// TwinCAT 3 PLC project CustomGenericDataType
// Title: TwinCAT Custom Generic Data Types
// Company: FisoThemes
// Author: Goodwill Mzumala
// ProjectVersion: 1.0.0.0
// Description: Library created to handle data in TwinCAT generically. Useful for overloading or creating multitype arrays.
// ProgramVersion: 3.1.4023.0
// libraries:
//   Tc2_Standard, * (Beckhoff Automation GmbH)
//   Tc2_System, * (Beckhoff Automation GmbH)
//   Tc3_Module, * (Beckhoff Automation GmbH)
// project tree:
//   DUTs/ ST_Arg_Pointer.TcDUT, ST_Arg.TcDUT
//   / PlcTask.TcTTO
//   POUs/Arguments/Bit/ F_BYTE_ARG.TcPOU, F_DWORD_ARG.TcPOU, F_LWORD_ARG.TcPOU, F_WORD_ARG.TcPOU
//   POUs/Arguments/Date/ F_DATE_ARG.TcPOU, F_DT_ARG.TcPOU, F_TOD_ARG.TcPOU
//   POUs/Arguments/Int/ F_DINT_ARG.TcPOU, F_INT_ARG.TcPOU, F_LINT_ARG.TcPOU, F_SINT_ARG.TcPOU, F_UDINT_ARG.TcPOU, F_UINT_ARG.TcPOU, F_ULINT_ARG.TcPOU, F_USINT_ARG.TcPOU
//   POUs/Arguments/Other/ F_ANY_ARG.TcPOU, F_PVOID_ARG.TcPOU
//   POUs/Arguments/Real/ F_LREAL_ARG.TcPOU, F_REAL_ARG.TcPOU
//   POUs/Arguments/String/ F_STRING_ARG.TcPOU, F_WSTRING_ARG.TcPOU
//   POUs/Arguments/Time/ F_LTIME_ARG.TcPOU, F_TIME_ARG.TcPOU
//   POUs/Examples/Example 1 - Generic Use Case/ P_Example_1.TcPOU
//   POUs/Examples/Example 2 - Dynamic Array Use Case/Files/ FB_Dynamic_Array.TcPOU, T_DynamicArrayDataType.TcDUT
//   POUs/Examples/Example 2 - Dynamic Array Use Case/ P_Example_2.TcPOU
//   POUs/ MAIN.TcPOU
//   POUs/Return Values/Bit/ F_BYTE_RTN.TcPOU, F_DWORD_RTN.TcPOU, F_LWORD_RTN.TcPOU, F_WORD_RTN.TcPOU
//   POUs/Return Values/Date/ F_DATE_RTN.TcPOU, F_DT_RTN.TcPOU, F_TOD_RTN.TcPOU
//   POUs/Return Values/Int/ F_DINT_RTN.TcPOU, F_INT_RTN.TcPOU, F_LINT_RTN.TcPOU, F_SINT_RTN.TcPOU, F_UDINT_RTN.TcPOU, F_UINT_RTN.TcPOU, F_ULINT_RTN.TcPOU, F_USINT_RTN.TcPOU
//   POUs/Return Values/Other/ F_PVOID_RTN.TcPOU
//   POUs/Return Values/Real/ F_LREAL_RTN.TcPOU, F_REAL_RTN.TcPOU
//   POUs/Return Values/String/ F_STRING_RTN.TcPOU, F_WSTRING_RTN.TcPOU
//   POUs/Return Values/Time/ F_LTIME_RTN.TcPOU, F_TIME_RTN.TcPOU
// real-time tasks:
//   TASK PlcTask: cycle T#10ms, priority 20, ADS port 350

CONFIGURATION CustomGenericDataType
    RESOURCE PLC ON TwinCAT3
        TASK PlcTask(INTERVAL := T#10ms, PRIORITY := 20);
        PROGRAM MAIN WITH PlcTask : MAIN;
    END_RESOURCE
END_CONFIGURATION

// ---- DUTs/ST_Arg_Pointer.TcDUT
(* Collection of pointers for F_ANY_ARG. *)
TYPE INTERNAL ST_Arg_Pointer :
STRUCT
    pBool			: POINTER TO BOOL;
    pByte			: POINTER TO BYTE;
    pWord			: POINTER TO WORD;
    pDWord			: POINTER TO DWORD;
    pLWord			: POINTER TO LWORD;
    pSint			: POINTER TO SINT;
    pInt			: POINTER TO INT;
    pDint			: POINTER TO DINT;
    pLint			: POINTER TO LINT;
    pUSint			: POINTER TO USINT;
    pUInt			: POINTER TO UINT;
    pUDint			: POINTER TO UDINT;
    pULint			: POINTER TO ULINT;
    pReal			: POINTER TO REAL;
    pLReal			: POINTER TO LREAL;
    pString			: POINTER TO STRING;
    pWString		: POINTER TO WSTRING;
    pTime			: POINTER TO TIME;
    pDate			: POINTER TO DATE;
    pDate_And_Time	: POINTER TO DATE_AND_TIME;
    pTime_Of_Day	: POINTER TO TIME_OF_DAY;
    pPointer		: PVOID;
	pLTime 			: POINTER TO LTIME;
END_STRUCT
END_TYPE

// ---- DUTs/ST_Arg.TcDUT
(* Generic data type used for Programs/Functions/Function Blocks. *)
TYPE ST_Arg EXTENDS __SYSTEM.AnyType :
STRUCT
	sValue : T_MaxString; 	// Data of parameter as a string for easy convertion.
END_STRUCT
END_TYPE

// ---- POUs/Examples/Example 2 - Dynamic Array Use Case/Files/T_DynamicArrayDataType.TcDUT
TYPE T_DynamicArrayDataType : ST_Arg; END_TYPE

// ---- POUs/MAIN.TcPOU
PROGRAM MAIN
VAR
	
END_VAR

P_Example_1();
P_Example_2();

END_PROGRAM

// ---- POUs/Examples/Example 1 - Generic Use Case/P_Example_1.TcPOU
PROGRAM P_Example_1
VAR
	stArg 	: ARRAY[0..5] OF ST_Arg;
	
	Numeric_Type 		: INT := 20;
	User_Defined_Type	: TON := (PT := T#10S);
	
	rtnInteger 	: INT;
	rtnPointer 	: POINTER TO TON;
	
END_VAR

// Store 
stArg[0] := F_ANY_ARG(Numeric_Type);
stArg[1] := F_INT_ARG(1);
stArg[2] := F_REAL_ARG(12.442);
stArg[3] := F_STRING_ARG('Cats');
stArg[4] := F_PVOID_ARG(ADR(User_Defined_Type));

rtnInteger := F_INT_RTN(stArg[0]);
rtnPointer := F_PVOID_RTN(stArg[4]);

END_PROGRAM

// ---- POUs/Arguments/Other/F_ANY_ARG.TcPOU
FUNCTION F_ANY_ARG : ST_Arg
VAR_INPUT
	Input : ANY;
END_VAR
VAR
	stArg 			: ST_Arg;
	stArg_Pointer 	: ST_Arg_Pointer;
	sysVar_Info 	: __SYSTEM.VAR_INFO;
END_VAR

stArg.TypeClass := Input.TypeClass;
stArg.pValue 	:= Input.pValue;
stArg.diSize 	:= Input.diSize;

CASE Input.TypeClass OF 
	__SYSTEM.TYPE_CLASS.TYPE_BOOL:
		stArg_Pointer.pBool := Input.pValue;
		stArg.sValue := TO_STRING(stArg_Pointer.pBool^);
		
    __SYSTEM.TYPE_CLASS.TYPE_BYTE:
		stArg_Pointer.pByte := Input.pValue;
		stArg.sValue := TO_STRING(stArg_Pointer.pByte^);
		
    __SYSTEM.TYPE_CLASS.TYPE_WORD:
		stArg_Pointer.pWord := Input.pValue;
		stArg.sValue := TO_STRING(stArg_Pointer.pWord^);
		
    __SYSTEM.TYPE_CLASS.TYPE_DWORD:
		stArg_Pointer.pDWord := Input.pValue;
		stArg.sValue := TO_STRING(stArg_Pointer.pDWord^);
		
    __SYSTEM.TYPE_CLASS.TYPE_LWORD:
		stArg_Pointer.pLWord := Input.pValue;
		stArg.sValue := TO_STRING(stArg_Pointer.pLWord^);
		
    __SYSTEM.TYPE_CLASS.TYPE_SINT:
		stArg_Pointer.pSint := Input.pValue;
		stArg.sValue := TO_STRING(stArg_Pointer.pSint^);
		
    __SYSTEM.TYPE_CLASS.TYPE_INT:
		stArg_Pointer.pInt := Input.pValue;
		stArg.sValue := TO_STRING(stArg_Pointer.pInt^);
		
    __SYSTEM.TYPE_CLASS.TYPE_DINT:
		stArg_Pointer.pDint := Input.pValue;
		stArg.sValue := TO_STRING(stArg_Pointer.pDint^);
		
    __SYSTEM.TYPE_CLASS.TYPE_LINT:
		stArg_Pointer.pLint := Input.pValue;
		stArg.sValue := TO_STRING(stArg_Pointer.pLint^);
		
    __SYSTEM.TYPE_CLASS.TYPE_USINT:
		stArg_Pointer.pUSint := Input.pValue;
		stArg.sValue := TO_STRING(stArg_Pointer.pUSint^);
		
    __SYSTEM.TYPE_CLASS.TYPE_UINT:
		stArg_Pointer.pUInt := Input.pValue;
		stArg.sValue := TO_STRING(stArg_Pointer.pUInt^);
		
    __SYSTEM.TYPE_CLASS.TYPE_UDINT:
		stArg_Pointer.pUDint := Input.pValue;
		stArg.sValue := TO_STRING(stArg_Pointer.pUDint^);
		
    __SYSTEM.TYPE_CLASS.TYPE_ULINT:
		stArg_Pointer.pULint := Input.pValue;
		stArg.sValue := TO_STRING(stArg_Pointer.pULint^);
		
   __SYSTEM.TYPE_CLASS.TYPE_REAL:
		stArg_Pointer.pReal := Input.pValue;
		stArg.sValue := TO_STRING(stArg_Pointer.pReal^);
		
    __SYSTEM.TYPE_CLASS.TYPE_LREAL:
		stArg_Pointer.pLReal := Input.pValue;
		stArg.sValue := TO_STRING(stArg_Pointer.pLReal^);
		
    __SYSTEM.TYPE_CLASS.TYPE_STRING:
		stArg_Pointer.pString := Input.pValue;
		stArg.sValue := TO_STRING(stArg_Pointer.pString^);
		
   __SYSTEM.TYPE_CLASS.TYPE_WSTRING:
		stArg_Pointer.pWString := Input.pValue;
		stArg.sValue := TO_STRING(stArg_Pointer.pWString^);
		
    __SYSTEM.TYPE_CLASS.TYPE_TIME:
		stArg_Pointer.pTime := Input.pValue;
		stArg.sValue := TO_STRING(stArg_Pointer.pTime^);
		
    __SYSTEM.TYPE_CLASS.TYPE_DATE:
		stArg_Pointer.pDate := Input.pValue;
		stArg.sValue := TO_STRING(stArg_Pointer.pDate^);
		
    __SYSTEM.TYPE_CLASS.TYPE_DATEANDTIME:
		stArg_Pointer.pDate_And_Time := Input.pValue;
		stArg.sValue := TO_STRING(stArg_Pointer.pDate_And_Time^);
		
    __SYSTEM.TYPE_CLASS.TYPE_TIMEOFDAY:
		stArg_Pointer.pTime_Of_Day := Input.pValue;
		stArg.sValue := TO_STRING(stArg_Pointer.pTime_Of_Day^);
	
	__SYSTEM.TYPE_CLASS.TYPE_POINTER:
		stArg.sValue := TO_STRING(Input.pValue);
		
	__SYSTEM.TYPE_CLASS.TYPE_LTIME:
		stArg_Pointer.pLTime := Input.pValue;
		stArg.sValue := TO_STRING(stArg_Pointer.pLTime^);
ELSE
	stArg.sValue := 'NULL'; 
END_CASE

F_ANY_ARG := stArg;

END_FUNCTION

// ---- POUs/Arguments/Int/F_INT_ARG.TcPOU
FUNCTION F_INT_ARG : ST_Arg
VAR_INPUT
	nInput : INT;
END_VAR
VAR
	stArg : ST_Arg;
	sysVar_Info : __SYSTEM.VAR_INFO;
END_VAR

sysVar_Info 	:= __VARINFO(nInput);
stArg.TypeClass := sysVar_Info.TypeClass;
stArg.pValue 	:= 0;
stArg.diSize 	:= SIZEOF(nInput);
stArg.sValue 	:= TO_STRING(nInput); 
F_INT_ARG := stArg;

END_FUNCTION

// ---- POUs/Arguments/Real/F_REAL_ARG.TcPOU
FUNCTION F_REAL_ARG : ST_Arg
VAR_INPUT
	fInput : REAL;
END_VAR
VAR
	stArg : ST_Arg;
	sysVar_Info : __SYSTEM.VAR_INFO;
END_VAR

sysVar_Info 	:= __VARINFO(fInput);
stArg.TypeClass := sysVar_Info.TypeClass;
stArg.pValue 	:= 0;
stArg.diSize 	:= SIZEOF(fInput);
stArg.sValue 	:= TO_STRING(fInput); 
F_REAL_ARG := stArg;

END_FUNCTION

// ---- POUs/Arguments/String/F_STRING_ARG.TcPOU
FUNCTION F_STRING_ARG : ST_Arg
VAR_INPUT
	sInput : T_MaxString;
END_VAR
VAR
	stArg : ST_Arg;
	sysVar_Info : __SYSTEM.VAR_INFO;
END_VAR

sysVar_Info 	:= __VARINFO(sInput);
stArg.TypeClass := sysVar_Info.TypeClass;
stArg.pValue 	:= 0;
stArg.diSize 	:= SIZEOF(sInput);
stArg.sValue 	:= sInput; 
F_STRING_ARG := stArg;

END_FUNCTION

// ---- POUs/Arguments/Other/F_PVOID_ARG.TcPOU
FUNCTION F_PVOID_ARG : ST_Arg
VAR_INPUT
	pInput : PVOID;
END_VAR
VAR
	stArg : ST_Arg;
	sysVar_Info : __SYSTEM.VAR_INFO;
END_VAR

sysVar_Info 	:= __VARINFO(pInput);
stArg.TypeClass := sysVar_Info.TypeClass;
stArg.pValue 	:= pInput;
stArg.diSize 	:= SIZEOF(pInput);
stArg.sValue 	:= TO_STRING(pInput); 
F_PVOID_ARG := stArg;

END_FUNCTION

// ---- POUs/Return Values/Int/F_INT_RTN.TcPOU
FUNCTION F_INT_RTN : INT
VAR_INPUT
	stArg : ST_Arg;
END_VAR
VAR
	sysVar_Info : __SYSTEM.VAR_INFO;
END_VAR

sysVar_Info := __VARINFO(F_INT_RTN);
IF stArg.TypeClass = sysVar_Info.TypeClass THEN 
	F_INT_RTN := TO_INT(stArg.sValue);
	END_IF

END_FUNCTION

// ---- POUs/Return Values/Other/F_PVOID_RTN.TcPOU
FUNCTION F_PVOID_RTN : PVOID
VAR_INPUT
	stArg : ST_Arg;
END_VAR
VAR_STAT
	sysVar_Info : __SYSTEM.VAR_INFO;
END_VAR

sysVar_Info := __VARINFO(F_PVOID_RTN);
IF stArg.TypeClass = sysVar_Info.TypeClass THEN 
	F_PVOID_RTN := stArg.pValue;
	END_IF

END_FUNCTION

// ---- POUs/Examples/Example 2 - Dynamic Array Use Case/P_Example_2.TcPOU
PROGRAM P_Example_2
VAR
	bIs_Empty, bInsert, bAdd, bfAccess, bnAccess, bsAccess, bResize, bClear : BOOL;
	fbDyn_Array : FB_Dynamic_Array(10);
	aArray 		: ARRAY[0..30] OF T_DynamicArrayDataType;
	nDyn_Size 	: DINT;
	
	fAccess 	: REAL; 
	nAccess 	: DINT; 
	sAccess 	: STRING; 
 
	i 			: DINT;
END_VAR

bIs_Empty := fbDyn_Array.Is_Empty();
nDyn_Size := fbDyn_Array.Size();
fbDyn_Array.Show(aArray);

IF bInsert THEN
	fbDyn_Array.Insert(F_STRING_ARG('FIRST'),0); 
	FOR i := 1 TO 9 DO fbDyn_Array.Insert(F_DINT_ARG(i*11),i); END_FOR
	bInsert := 0;
	END_IF

IF bAdd 	THEN fbDyn_Array.Insert(F_REAL_ARG(33.33),10); 	bAdd 	:= 0; END_IF
IF bfAccess THEN fAccess := F_REAL_RTN(fbDyn_Array.Access(10)); bfAccess := 0; END_IF
IF bnAccess THEN nAccess := F_DINT_RTN(fbDyn_Array.Access(2)); bnAccess := 0; END_IF
IF bsAccess THEN sAccess := F_STRING_RTN(fbDyn_Array.Access(0)); bsAccess := 0; END_IF
IF bResize 	THEN fbDyn_Array.Resize(5); bResize := 0; END_IF
IF bClear 	THEN fbDyn_Array.Clear(); bClear := 0; END_IF

END_PROGRAM

// ---- POUs/Examples/Example 2 - Dynamic Array Use Case/Files/FB_Dynamic_Array.TcPOU
FUNCTION_BLOCK FB_Dynamic_Array
VAR_INPUT
	
END_VAR
VAR_OUTPUT
END_VAR
VAR
	pData 	: POINTER TO T_DynamicArrayDataType;
	nLength : DINT;
	t_Null	: T_DynamicArrayDataType := (TypeClass := __SYSTEM.TYPE_CLASS.TYPE_NONE, pValue := 0 , diSize := -1, sValue := 'NULL');
END_VAR

(* Get element in array from specified poisiton. *)
METHOD Access : T_DynamicArrayDataType
VAR_INPUT
	nPosition : DINT;  // Position of element in dynamic array, 0 indexed.
END_VAR
IF nPosition < 0 THEN Access := t_Null; RETURN; END_IF
IF THIS^.Is_Empty() THEN FB_Init(FALSE,FALSE,(nPosition+1)*2); END_IF
IF nPosition >= THIS^.Size() THEN THIS^.Insert(t_Null, nPosition); END_IF
Access := THIS^.pData[nPosition];
END_METHOD

(* Deletes array from memory. *)
METHOD Clear
VAR_INPUT
END_VAR
IF NOT(THIS^.Is_Empty()) THEN __DELETE(THIS^.pData); THIS^.Is_Empty(); END_IF
END_METHOD

METHOD FB_exit : BOOL
VAR_INPUT
	bInCopyCode : BOOL; // if TRUE, the exit method is called for exiting an instance that is copied afterwards (online change).
END_VAR
THIS^.Clear();
END_METHOD

METHOD FB_init : BOOL
VAR_INPUT
	bInitRetains 	: BOOL; 	// if TRUE, the retain variables are initialized (warm start / cold start)
	bInCopyCode 	: BOOL;  	// if TRUE, the instance afterwards gets moved into the copy code (online change)
	nLength 		: DINT; 	// Length to initialize array with, default is 10;
END_VAR
THIS^.Clear();
IF nLength > 0 THEN 
	THIS^.pData := __NEW(BYTE, TO_UDINT(SIZEOF(T_DynamicArrayDataType)*nLength)); 
	END_IF
THIS^.nLength := nLength;
END_METHOD

(* Insert element into array at specified position. *)
METHOD Insert
VAR_INPUT
	Data 		: T_DynamicArrayDataType; 	// Data to insert in dynamic array.
	nPosition 	: DINT; 					// Position to insert data at in the dynamic array, 0 indexed. 
END_VAR
VAR
	pTemp_Data 		: POINTER TO T_DynamicArrayDataType;
	nTemp_Length 	: DINT;
	i : DINT;
END_VAR
IF nPosition < 0 THEN RETURN; END_IF
IF THIS^.Is_Empty() THEN FB_Init(FALSE,FALSE,(nPosition+1)*2); END_IF
IF nPosition < THIS^.Size() THEN 
	THIS^.pData[nPosition] := Data;
ELSE 
	THIS^.Resize((nPosition+1)*2);
	THIS^.pData[nPosition] := Data;
	END_IF
END_METHOD

(* Checks if array is empty. *)
METHOD Is_Empty : BOOL
VAR_INPUT
END_VAR
Is_Empty := THIS^.pData = 0;
IF Is_Empty THEN THIS^.nLength := 0; END_IF
END_METHOD

(* Manually resize dynamic array length. If Array become smaller, elements higher positions will be deleted. *)
METHOD Resize
VAR_INPUT
	nLength : DINT; // New length of dynamic array.
END_VAR
VAR
	pTemp_Data 		: POINTER TO T_DynamicArrayDataType;
	nTemp_Length 	: DINT;
	i : DINT;
END_VAR
IF nLength <= 0 THEN THIS^.Clear(); RETURN; END_IF
IF THIS^.Is_Empty() THEN FB_init(FALSE,FALSE,nLength); RETURN; END_IF
IF THIS^.nLength = nLength THEN RETURN; END_IF

pTemp_Data 		:= THIS^.pData; 

nTemp_Length 	:= THIS^.nLength;
THIS^.nLength 	:= nLength;

THIS^.pData := __NEW(BYTE, TO_UDINT(SIZEOF(T_DynamicArrayDataType)*THIS^.nLength));
FOR i := 0 TO TO_DINT(nTemp_Length-1) DO 
	IF i > TO_DINT(THIS^.nLength-1) THEN EXIT; END_IF 
	THIS^.pData[i] := pTemp_Data[i]; 
	END_FOR
__DELETE(pTemp_Data);
END_METHOD

(* Display elements in dynamic array in a static array. *)
METHOD Show
VAR_IN_OUT
	aList : ARRAY[*] OF T_DynamicArrayDataType; // Static array to display data in dynamic array.
END_VAR
VAR
	i,j : DINT; 
END_VAR
FOR i := LOWER_BOUND(aList, 1) TO UPPER_BOUND(aList, 1) DO
	IF (j < TO_DINT(THIS^.Size())) AND NOT(THIS^.Is_Empty()) THEN
		aList[i] := THIS^.pData[j];
		j := j + 1; 
	ELSE 
		aList[i] := t_Null;
	 	END_IF
	END_FOR
END_METHOD

(* Gets the length of dynamic array. *)
METHOD Size : DINT
VAR_INPUT
END_VAR
Is_Empty(); Size := THIS^.nLength;
END_METHOD

END_FUNCTION_BLOCK

// ---- POUs/Arguments/Int/F_DINT_ARG.TcPOU
FUNCTION F_DINT_ARG : ST_Arg
VAR_INPUT
	nInput : DINT;
END_VAR
VAR
	stArg : ST_Arg;
	sysVar_Info : __SYSTEM.VAR_INFO;
END_VAR

sysVar_Info := __VARINFO(nInput);
stArg.TypeClass := sysVar_Info.TypeClass;
stArg.pValue 	:= 0;
stArg.diSize 	:= SIZEOF(nInput);
stArg.sValue 	:= TO_STRING(nInput); 
F_DINT_ARG := stArg;

END_FUNCTION

// ---- POUs/Return Values/Real/F_REAL_RTN.TcPOU
FUNCTION F_REAL_RTN : REAL
VAR_INPUT
	stArg : ST_Arg;
END_VAR
VAR
	sysVar_Info : __SYSTEM.VAR_INFO;
END_VAR

sysVar_Info := __VARINFO(F_REAL_RTN);
IF stArg.TypeClass = sysVar_Info.TypeClass THEN 
	F_REAL_RTN := TO_REAL(stArg.sValue);
	END_IF

END_FUNCTION

// ---- POUs/Return Values/Int/F_DINT_RTN.TcPOU
FUNCTION F_DINT_RTN : DINT
VAR_INPUT
	stArg : ST_Arg;
END_VAR
VAR
	sysVar_Info : __SYSTEM.VAR_INFO;
END_VAR

sysVar_Info := __VARINFO(F_DINT_RTN);
IF stArg.TypeClass = sysVar_Info.TypeClass THEN 
	F_DINT_RTN := TO_DINT(stArg.sValue);
	END_IF

END_FUNCTION

// ---- POUs/Return Values/String/F_STRING_RTN.TcPOU
FUNCTION F_STRING_RTN : T_MaxString
VAR_INPUT
	stArg : ST_Arg;
END_VAR
VAR
	sysVar_Info : __SYSTEM.VAR_INFO;
END_VAR

sysVar_Info := __VARINFO(F_STRING_RTN);
IF stArg.TypeClass = sysVar_Info.TypeClass THEN 
	F_STRING_RTN := TO_STRING(stArg.sValue);
	END_IF

END_FUNCTION

// ---- POUs/Arguments/Bit/F_BYTE_ARG.TcPOU
FUNCTION F_BYTE_ARG : ST_Arg
VAR_INPUT
	nInput : BYTE;
END_VAR
VAR
	stArg : ST_Arg;
	sysVar_Info : __SYSTEM.VAR_INFO;
END_VAR

sysVar_Info 	:= __VARINFO(nInput);
stArg.TypeClass := sysVar_Info.TypeClass;
stArg.pValue 	:= 0;
stArg.diSize 	:= SIZEOF(nInput);
stArg.sValue 	:= TO_STRING(nInput);
F_BYTE_ARG := stArg;

END_FUNCTION

// ---- POUs/Arguments/Bit/F_DWORD_ARG.TcPOU
FUNCTION F_DWORD_ARG : ST_Arg
VAR_INPUT
	dwInput : DWORD;
END_VAR
VAR
	stArg : ST_Arg;
	sysVar_Info : __SYSTEM.VAR_INFO;
END_VAR

sysVar_Info 	:= __VARINFO(dwInput);
stArg.TypeClass := sysVar_Info.TypeClass;
stArg.pValue 	:= 0;
stArg.diSize 	:= SIZEOF(dwInput);
stArg.sValue 	:= TO_STRING(dwInput); 
F_DWORD_ARG := stArg;

END_FUNCTION

// ---- POUs/Arguments/Bit/F_LWORD_ARG.TcPOU
FUNCTION F_LWORD_ARG : ST_Arg
VAR_INPUT
	lwInput : LWORD;
END_VAR
VAR
	stArg : ST_Arg;
	sysVar_Info : __SYSTEM.VAR_INFO;
END_VAR

sysVar_Info 	:= __VARINFO(lwInput);
stArg.TypeClass := sysVar_Info.TypeClass;
stArg.pValue 	:= 0;
stArg.diSize 	:= SIZEOF(lwInput);
stArg.sValue 	:= TO_STRING(lwInput); 
F_LWORD_ARG := stArg;

END_FUNCTION

// ---- POUs/Arguments/Bit/F_WORD_ARG.TcPOU
FUNCTION F_WORD_ARG : ST_Arg
VAR_INPUT
	wInput : WORD;
END_VAR
VAR
	stArg : ST_Arg;
	sysVar_Info : __SYSTEM.VAR_INFO;
END_VAR

sysVar_Info 	:= __VARINFO(wInput);
stArg.TypeClass := sysVar_Info.TypeClass;
stArg.pValue 	:= 0;
stArg.diSize 	:= SIZEOF(wInput);
stArg.sValue 	:= TO_STRING(wInput); 
F_WORD_ARG := stArg;

END_FUNCTION

// ---- POUs/Arguments/Date/F_DATE_ARG.TcPOU
FUNCTION F_DATE_ARG : ST_Arg
VAR_INPUT
	dtInput : DATE;
END_VAR
VAR
	stArg : ST_Arg;
	sysVar_Info : __SYSTEM.VAR_INFO;
END_VAR

sysVar_Info 	:= __VARINFO(dtInput);
stArg.TypeClass := sysVar_Info.TypeClass;
stArg.pValue 	:= 0;
stArg.diSize 	:= SIZEOF(dtInput);
stArg.sValue 	:= TO_STRING(dtInput); 
F_DATE_ARG := stArg;

END_FUNCTION

// ---- POUs/Arguments/Date/F_DT_ARG.TcPOU
FUNCTION F_DT_ARG : ST_Arg
VAR_INPUT
	dtInput : DT;
END_VAR
VAR
	stArg : ST_Arg;
	sysVar_Info : __SYSTEM.VAR_INFO;
END_VAR

sysVar_Info 	:= __VARINFO(dtInput);
stArg.TypeClass := sysVar_Info.TypeClass;
stArg.pValue 	:= 0;
stArg.diSize 	:= SIZEOF(dtInput);
stArg.sValue 	:= TO_STRING(dtInput); 
THIS^ := stArg;

END_FUNCTION

// ---- POUs/Arguments/Date/F_TOD_ARG.TcPOU
FUNCTION F_TOD_ARG : ST_Arg
VAR_INPUT
	todInput : TOD;
END_VAR
VAR
	stArg : ST_Arg;
	sysVar_Info : __SYSTEM.VAR_INFO;
END_VAR

sysVar_Info 	:= __VARINFO(todInput);
stArg.TypeClass := sysVar_Info.TypeClass;
stArg.pValue 	:= 0;
stArg.diSize 	:= SIZEOF(todInput);
stArg.sValue 	:= TO_STRING(todInput); 
F_TOD_ARG := stArg;

END_FUNCTION

// ---- POUs/Arguments/Int/F_LINT_ARG.TcPOU
FUNCTION F_LINT_ARG : ST_Arg
VAR_INPUT
	nInput : LINT;
END_VAR
VAR
	stArg : ST_Arg;
	sysVar_Info : __SYSTEM.VAR_INFO;
END_VAR

sysVar_Info 	:= __VARINFO(nInput);
stArg.TypeClass := sysVar_Info.TypeClass;
stArg.pValue 	:= 0;
stArg.diSize 	:= SIZEOF(nInput);
stArg.sValue 	:= TO_STRING(nInput); 
F_LINT_ARG := stArg;

END_FUNCTION

// ---- POUs/Arguments/Int/F_SINT_ARG.TcPOU
FUNCTION F_SINT_ARG : ST_Arg
VAR_INPUT
	nInput : SINT;
END_VAR
VAR
	stArg : ST_Arg;
	sysVar_Info : __SYSTEM.VAR_INFO;
END_VAR

sysVar_Info 	:= __VARINFO(nInput);
stArg.TypeClass := sysVar_Info.TypeClass;
stArg.pValue 	:= 0;
stArg.diSize 	:= SIZEOF(nInput);
stArg.sValue 	:= TO_STRING(nInput); 
F_SINT_ARG := stArg;

END_FUNCTION

// ---- POUs/Arguments/Int/F_UDINT_ARG.TcPOU
FUNCTION F_UDINT_ARG : ST_Arg
VAR_INPUT
	nInput : UDINT;
END_VAR
VAR
	stArg : ST_Arg;
	sysVar_Info : __SYSTEM.VAR_INFO;
END_VAR

sysVar_Info := __VARINFO(nInput);
stArg.TypeClass := sysVar_Info.TypeClass;
stArg.pValue 	:= 0;
stArg.diSize 	:= SIZEOF(nInput);
stArg.sValue 	:= TO_STRING(nInput); 
F_UDINT_ARG := stArg;

END_FUNCTION

// ---- POUs/Arguments/Int/F_UINT_ARG.TcPOU
FUNCTION F_UINT_ARG : ST_Arg
VAR_INPUT
	nInput : UINT;
END_VAR
VAR
	stArg : ST_Arg;
	sysVar_Info : __SYSTEM.VAR_INFO;
END_VAR

sysVar_Info 	:= __VARINFO(nInput);
stArg.TypeClass := sysVar_Info.TypeClass;
stArg.pValue 	:= 0;
stArg.diSize 	:= SIZEOF(nInput);
stArg.sValue 	:= TO_STRING(nInput); 
F_UINT_ARG := stArg;

END_FUNCTION

// ---- POUs/Arguments/Int/F_ULINT_ARG.TcPOU
FUNCTION F_ULINT_ARG : ST_Arg
VAR_INPUT
	nInput : ULINT;
END_VAR
VAR
	stArg : ST_Arg;
	sysVar_Info : __SYSTEM.VAR_INFO;
END_VAR

sysVar_Info 	:= __VARINFO(nInput);
stArg.TypeClass := sysVar_Info.TypeClass;
stArg.pValue 	:= 0;
stArg.diSize 	:= SIZEOF(nInput);
stArg.sValue 	:= TO_STRING(nInput); 
F_ULINT_ARG := stArg;

END_FUNCTION

// ---- POUs/Arguments/Int/F_USINT_ARG.TcPOU
FUNCTION F_USINT_ARG : ST_Arg
VAR_INPUT
	nInput : USINT;
END_VAR
VAR
	stArg : ST_Arg;
	sysVar_Info : __SYSTEM.VAR_INFO;
END_VAR

sysVar_Info 	:= __VARINFO(nInput);
stArg.TypeClass := sysVar_Info.TypeClass;
stArg.pValue 	:= 0;
stArg.diSize 	:= SIZEOF(nInput);
stArg.sValue 	:= TO_STRING(nInput); 
F_USINT_ARG := stArg;

END_FUNCTION

// ---- POUs/Arguments/Real/F_LREAL_ARG.TcPOU
FUNCTION F_LREAL_ARG : ST_Arg
VAR_INPUT
	fInput : LREAL;
END_VAR
VAR
	stArg : ST_Arg;
	sysVar_Info : __SYSTEM.VAR_INFO;
END_VAR

sysVar_Info 	:= __VARINFO(fInput);
stArg.TypeClass := sysVar_Info.TypeClass;
stArg.pValue 	:= 0;
stArg.diSize 	:= SIZEOF(fInput);
stArg.sValue 	:= TO_STRING(fInput); 
F_LREAL_ARG := stArg;

END_FUNCTION

// ---- POUs/Arguments/String/F_WSTRING_ARG.TcPOU
FUNCTION F_WSTRING_ARG : ST_Arg
VAR_INPUT
	wsInput : WSTRING(255);
END_VAR
VAR
	stArg : ST_Arg;
	sysVar_Info : __SYSTEM.VAR_INFO;
END_VAR

sysVar_Info 	:= __VARINFO(wsInput);
stArg.TypeClass := sysVar_Info.TypeClass;
stArg.pValue 	:= 0;
stArg.diSize 	:= SIZEOF(wsInput);
stArg.sValue 	:= TO_STRING(wsInput); 
F_WSTRING_ARG := stArg;

END_FUNCTION

// ---- POUs/Arguments/Time/F_LTIME_ARG.TcPOU
FUNCTION F_LTIME_ARG : ST_Arg
VAR_INPUT
	tInput : LTIME;
END_VAR
VAR
	stArg : ST_Arg;
	sysVar_Info : __SYSTEM.VAR_INFO;
END_VAR

sysVar_Info 	:= __VARINFO(tInput);
stArg.TypeClass := sysVar_Info.TypeClass;
stArg.pValue 	:= 0;
stArg.diSize 	:= SIZEOF(tInput);
stArg.sValue 	:= TO_STRING(tInput); 
F_LTIME_ARG := stArg;

END_FUNCTION

// ---- POUs/Arguments/Time/F_TIME_ARG.TcPOU
FUNCTION F_TIME_ARG : ST_Arg
VAR_INPUT
	tInput : TIME;
END_VAR
VAR
	stArg : ST_Arg;
	sysVar_Info : __SYSTEM.VAR_INFO;
END_VAR

sysVar_Info 	:= __VARINFO(tInput);
stArg.TypeClass := sysVar_Info.TypeClass;
stArg.pValue 	:= 0;
stArg.diSize 	:= SIZEOF(tInput);
stArg.sValue 	:= TO_STRING(tInput); 
F_TIME_ARG := stArg;

END_FUNCTION

// ---- POUs/Return Values/Bit/F_BYTE_RTN.TcPOU
FUNCTION F_BYTE_RTN : BYTE
VAR_INPUT
	stArg : ST_Arg;
END_VAR
VAR
	sysVar_Info : __SYSTEM.VAR_INFO;
END_VAR

sysVar_Info := __VARINFO(F_BYTE_RTN);
IF stArg.TypeClass = sysVar_Info.TypeClass THEN 
	F_BYTE_RTN := TO_BYTE(stArg.sValue);
	END_IF

END_FUNCTION

// ---- POUs/Return Values/Bit/F_DWORD_RTN.TcPOU
FUNCTION F_DWORD_RTN : DWORD
VAR_INPUT
	stArg : ST_Arg;
END_VAR
VAR
	sysVar_Info : __SYSTEM.VAR_INFO;
END_VAR

sysVar_Info := __VARINFO(F_DWORD_RTN);
IF stArg.TypeClass = sysVar_Info.TypeClass THEN 
	F_DWORD_RTN := TO_DWORD(stArg.sValue);
	END_IF

END_FUNCTION

// ---- POUs/Return Values/Bit/F_LWORD_RTN.TcPOU
FUNCTION F_LWORD_RTN : LWORD
VAR_INPUT
	stArg : ST_Arg;
END_VAR
VAR
	sysVar_Info : __SYSTEM.VAR_INFO;
END_VAR

sysVar_Info := __VARINFO(F_LWORD_RTN);
IF stArg.TypeClass = sysVar_Info.TypeClass THEN 
	F_LWORD_RTN := TO_LWORD(stArg.sValue);
	END_IF

END_FUNCTION

// ---- POUs/Return Values/Bit/F_WORD_RTN.TcPOU
FUNCTION F_WORD_RTN : WORD
VAR_INPUT
	stArg : ST_Arg;
END_VAR
VAR
	sysVar_Info : __SYSTEM.VAR_INFO;
END_VAR

sysVar_Info := __VARINFO(F_WORD_RTN);
IF stArg.TypeClass = sysVar_Info.TypeClass THEN 
	F_WORD_RTN := TO_WORD(stArg.sValue);
	END_IF

END_FUNCTION

// ---- POUs/Return Values/Date/F_DATE_RTN.TcPOU
FUNCTION F_DATE_RTN : DATE
VAR_INPUT
	stArg : ST_Arg;
END_VAR
VAR
	sysVar_Info : __SYSTEM.VAR_INFO;
END_VAR

sysVar_Info := __VARINFO(F_DATE_RTN);
IF stArg.TypeClass = sysVar_Info.TypeClass THEN 
	F_DATE_RTN := TO_DATE(stArg.sValue);
	END_IF

END_FUNCTION

// ---- POUs/Return Values/Date/F_DT_RTN.TcPOU
FUNCTION F_DT_RTN : DT
VAR_INPUT
	stArg : ST_Arg;
END_VAR
VAR
	sysVar_Info : __SYSTEM.VAR_INFO;
END_VAR

sysVar_Info := __VARINFO(F_DT_RTN);
IF stArg.TypeClass = sysVar_Info.TypeClass THEN 
	F_DT_RTN := TO_DT(stArg.sValue);
	END_IF

END_FUNCTION

// ---- POUs/Return Values/Date/F_TOD_RTN.TcPOU
FUNCTION F_TOD_RTN : TOD
VAR_INPUT
	stArg : ST_Arg;
END_VAR
VAR
	sysVar_Info : __SYSTEM.VAR_INFO;
END_VAR

sysVar_Info := __VARINFO(F_TOD_RTN);
IF stArg.TypeClass = sysVar_Info.TypeClass THEN 
	F_TOD_RTN := TO_TOD(stArg.sValue);
	END_IF

END_FUNCTION

// ---- POUs/Return Values/Int/F_LINT_RTN.TcPOU
FUNCTION F_LINT_RTN : LINT
VAR_INPUT
	stArg : ST_Arg;
END_VAR
VAR
	sysVar_Info : __SYSTEM.VAR_INFO;
END_VAR

sysVar_Info := __VARINFO(F_LINT_RTN);
IF stArg.TypeClass = sysVar_Info.TypeClass THEN 
	F_LINT_RTN := TO_LINT(stArg.sValue);
	END_IF

END_FUNCTION

// ---- POUs/Return Values/Int/F_SINT_RTN.TcPOU
FUNCTION F_SINT_RTN : SINT
VAR_INPUT
	stArg : ST_Arg;
END_VAR
VAR
	sysVar_Info : __SYSTEM.VAR_INFO;
END_VAR

sysVar_Info := __VARINFO(F_SINT_RTN);
IF stArg.TypeClass = sysVar_Info.TypeClass THEN 
	F_SINT_RTN := TO_SINT(stArg.sValue);
	END_IF

END_FUNCTION

// ---- POUs/Return Values/Int/F_UDINT_RTN.TcPOU
FUNCTION F_UDINT_RTN : UDINT
VAR_INPUT
	stArg : ST_Arg;
END_VAR
VAR
	sysVar_Info : __SYSTEM.VAR_INFO;
END_VAR

sysVar_Info := __VARINFO(F_UDINT_RTN);
IF stArg.TypeClass = sysVar_Info.TypeClass THEN 
	F_UDINT_RTN := TO_UDINT(stArg.sValue);
	END_IF

END_FUNCTION

// ---- POUs/Return Values/Int/F_UINT_RTN.TcPOU
FUNCTION F_UINT_RTN : UINT
VAR_INPUT
	stArg : ST_Arg;
END_VAR
VAR
	sysVar_Info : __SYSTEM.VAR_INFO;
END_VAR

sysVar_Info := __VARINFO(F_UINT_RTN);
IF stArg.TypeClass = sysVar_Info.TypeClass THEN 
	F_UINT_RTN := TO_UINT(stArg.sValue);
	END_IF

END_FUNCTION

// ---- POUs/Return Values/Int/F_ULINT_RTN.TcPOU
FUNCTION F_ULINT_RTN : ULINT
VAR_INPUT
	stArg : ST_Arg;
END_VAR
VAR
	sysVar_Info : __SYSTEM.VAR_INFO;
END_VAR

sysVar_Info := __VARINFO(F_ULINT_RTN);
IF stArg.TypeClass = sysVar_Info.TypeClass THEN 
	F_ULINT_RTN := TO_ULINT(stArg.sValue);
	END_IF

END_FUNCTION

// ---- POUs/Return Values/Int/F_USINT_RTN.TcPOU
FUNCTION F_USINT_RTN : USINT
VAR_INPUT
	stArg : ST_Arg;
END_VAR
VAR
	sysVar_Info : __SYSTEM.VAR_INFO;
END_VAR

sysVar_Info := __VARINFO(F_USINT_RTN);
IF stArg.TypeClass = sysVar_Info.TypeClass THEN 
	F_USINT_RTN := TO_USINT(stArg.sValue);
	END_IF

END_FUNCTION

// ---- POUs/Return Values/Real/F_LREAL_RTN.TcPOU
FUNCTION F_LREAL_RTN : LREAL
VAR_INPUT
	stArg : ST_Arg;
END_VAR
VAR
	sysVar_Info : __SYSTEM.VAR_INFO;
END_VAR

sysVar_Info := __VARINFO(F_LREAL_RTN);
IF stArg.TypeClass = sysVar_Info.TypeClass THEN 
	F_LREAL_RTN := TO_LREAL(stArg.sValue);
	END_IF

END_FUNCTION

// ---- POUs/Return Values/String/F_WSTRING_RTN.TcPOU
FUNCTION F_WSTRING_RTN : WSTRING(255)
VAR_INPUT
	stArg : ST_Arg;
END_VAR
VAR
	sysVar_Info : __SYSTEM.VAR_INFO;
END_VAR

sysVar_Info := __VARINFO(F_WSTRING_RTN);
IF stArg.TypeClass = sysVar_Info.TypeClass THEN 
	F_WSTRING_RTN := TO_WSTRING(stArg.sValue);
	END_IF

END_FUNCTION

// ---- POUs/Return Values/Time/F_LTIME_RTN.TcPOU
FUNCTION F_LTIME_RTN : LTIME
VAR_INPUT
	stArg : ST_Arg;
END_VAR
VAR
	sysVar_Info : __SYSTEM.VAR_INFO;
END_VAR

sysVar_Info := __VARINFO(F_LTIME_RTN);
IF stArg.TypeClass = sysVar_Info.TypeClass THEN 
	F_LTIME_RTN := TO_LTIME(stArg.sValue);
	END_IF

END_FUNCTION

// ---- POUs/Return Values/Time/F_TIME_RTN.TcPOU
FUNCTION F_TIME_RTN : TIME
VAR_INPUT
	stArg : ST_Arg;
END_VAR
VAR
	sysVar_Info : __SYSTEM.VAR_INFO;
END_VAR

sysVar_Info := __VARINFO(F_TIME_RTN);
IF stArg.TypeClass = sysVar_Info.TypeClass THEN 
	F_TIME_RTN := TO_TIME(stArg.sValue);
	END_IF

END_FUNCTION
